Universal Robots PolyScope program: URClient.urp

Program URClient (createdIn=3.1.17195 lastSavedIn=3.2.19293 directory=/programs installation=default robotSerialNumber=2015351391)
Calibrated DH parameters: a=[0.000352, -0.161198, -0.373486, 0.00005, 0.000049, 0]; d=[0.089268, 352.477598, -320.08558, -32.281492, 0.094939, 0.082518]; alpha=[1.570728, 0.001116, -0.003686, 1.571189, -1.570572, 0]; deltaTheta=[-0.000012, 1.181849, -1.491165, 0.309495, -0.000007, 0.000025]
BeforeStart
  open := socket_open("192.168.1.6",5000)
  Loop While (checkContinuously=false) expression=open≟ False
    open := socket_open("192.168.1.6",5000)
  targetPos := p[0,0,0,0,0,0]
  counter := 6
Robot Program (runOnlyOnce=false motionType=MoveJ speed=1.047198 acceleration=1.396263 recalculateMotions=false)
  sendToServer :=  (valueSource=Operator message=send to server valueType=String)
  Script: socket_send_string(sendToServer)
  receiveFromServ := socket_read_ascii_float(6)
  Wait Sleep waitTime=10
  Loop While (checkContinuously=false) expression=receiveFromServ[0]≠6
    Wait Sleep waitTime=0.3
    receiveFromServ := socket_read_ascii_float(6)
  Loop While (checkContinuously=false) expression=counter<6
    Script: targetPos[counter]=receiveFromServ[counter+1]
    counter := counter+1
  MoveJ speed 60 deg/s, acceleration 80 deg/s^2 (recalculateMotions=false)
    Waypoint Waypoint (Variable): variable=targetPos
